FUNCTION_BLOCK Seq_Get_Part EXTENDS FB_Basis IMPLEMENTS I_Sequenz
VAR_INPUT
	// Skillzuweisung
	R_Move					:I_Skill_Roboter;
	G_Move					:I_Skill_SmartGreifer;
	
	// Prozessparameter		
	RobParam				:ARRAY[0..2] OF sRoboterProzessVariablen;
	GripParam				:ARRAY[0..1] OF sSmartGreiferProzessVariablen;
END_VAR
VAR_OUTPUT
END_VAR
VAR
	// Interne Sequenzen
	Seq_Ausrichten			:Seq_Ausrichten;
END_VAR

// Ablauf
ACT_Ablauf();

// Zustandshandling
CASE iState OF
	0:	// BEREIT
		IF bStart THEN
			iState := 1;
		END_IF
	1:	// LAUFEND
		IF eSysCommand = 4 THEN
			bReset := TRUE;
			SFCReset := TRUE;
		END_IF
		
		IF bBeendet OR bReset THEN
			bReset := FALSE;
			SFCReset := FALSE;
			iState := 0;
		END_IF
	2: // ABGESCHLOSSEN
		IF SFCCurrentStep = 'Init' THEN
			iState := 0;
		END_IF
END_CASE

ACTION ACT_Ablauf:
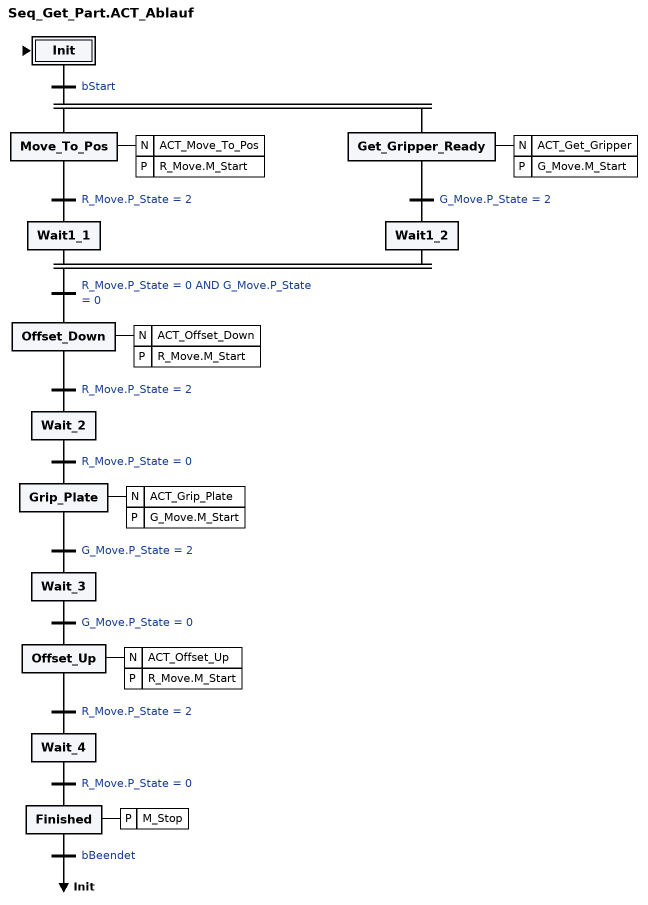
INITIAL_STEP Init:
END_STEP
TRANSITION FROM Init TO (Move_To_Pos, Get_Gripper_Ready)
    := bStart;
END_TRANSITION
STEP Move_To_Pos:
    ACT_Move_To_Pos(N);
    R_Move.M_Start(P);
END_STEP
TRANSITION FROM Move_To_Pos TO Wait1_1
    := R_Move.P_State = 2;
END_TRANSITION
STEP Wait1_1:
END_STEP
STEP Get_Gripper_Ready:
    ACT_Get_Gripper(N);
    G_Move.M_Start(P);
END_STEP
TRANSITION FROM Get_Gripper_Ready TO Wait1_2
    := G_Move.P_State = 2;
END_TRANSITION
STEP Wait1_2:
END_STEP
TRANSITION FROM (Wait1_1, Wait1_2) TO Offset_Down
    := R_Move.P_State = 0 AND G_Move.P_State = 0;
END_TRANSITION
STEP Offset_Down:
    ACT_Offset_Down(N);
    R_Move.M_Start(P);
END_STEP
TRANSITION FROM Offset_Down TO Wait_2
    := R_Move.P_State = 2;
END_TRANSITION
STEP Wait_2:
END_STEP
TRANSITION FROM Wait_2 TO Grip_Plate
    := R_Move.P_State = 0;
END_TRANSITION
STEP Grip_Plate:
    ACT_Grip_Plate(N);
    G_Move.M_Start(P);
END_STEP
TRANSITION FROM Grip_Plate TO Wait_3
    := G_Move.P_State = 2;
END_TRANSITION
STEP Wait_3:
END_STEP
TRANSITION FROM Wait_3 TO Offset_Up
    := G_Move.P_State = 0;
END_TRANSITION
STEP Offset_Up:
    ACT_Offset_Up(N);
    R_Move.M_Start(P);
END_STEP
TRANSITION FROM Offset_Up TO Wait_4
    := R_Move.P_State = 2;
END_TRANSITION
STEP Wait_4:
END_STEP
TRANSITION FROM Wait_4 TO Finished
    := R_Move.P_State = 0;
END_TRANSITION
STEP Finished:
    M_Stop(P);
END_STEP
TRANSITION FROM Finished TO Init
    := bBeendet;
END_TRANSITION
END_ACTION

ACTION ACT_Get_Gripper:
G_Move.P_SGripperParam := GripParam[0];
END_ACTION

ACTION ACT_Grip_Plate:
G_Move.P_SGripperParam := GripParam[1];
END_ACTION

ACTION ACT_Move_To_Pos:
R_Move.P_RobotParam := RobParam[0];
END_ACTION

ACTION ACT_Offset_Down:
R_Move.P_RobotParam := RobParam[1];
END_ACTION

ACTION ACT_Offset_Up:
R_Move.P_RobotParam := RobParam[2];
END_ACTION

END_FUNCTION_BLOCK

(* stored: Version 1.1.0.1
   POU Seq_Get_Part: Id {a8e83b85-49ec-4e2e-832d-d1ed2ea570f3}, SpecialFunc None
   Folder 01_Zuweisung: Id {663d7792-061a-4957-b277-18d59668cbbb}
   Action ACT_Ablauf: Id {7b69927b-4ec7-4216-99d9-848570b2aeda}
   Action ACT_Get_Gripper: Id {7c43d1d5-80ed-4978-86c1-f1210d3c12d5}
   Action ACT_Grip_Plate: Id {3c3d93b9-417a-4929-a117-05ba318880e4}
   Action ACT_Move_To_Pos: Id {89c2ffb9-97fa-482e-ad9a-c9705147f20a}
   Action ACT_Offset_Down: Id {18784caf-c27a-4702-9aa9-018a03b52983}
   Action ACT_Offset_Up: Id {69ebfc2c-44ed-43fe-a5df-2898fdda2428} *)
